FUNCTION_BLOCK FB_Holder
VAR_INPUT
	i_i_HolderPosition:	INT;
	Loaded:BOOL;
	Eingeschraubt	:	BOOL;
	Abgeschraubt: BOOL;
	Nagel: FB_Nagel;
END_VAR

METHOD MoveForward : BOOL
VAR_INPUT

END_VAR
i_i_HolderPosition:=i_i_HolderPosition+1;
END_METHOD

END_FUNCTION_BLOCK

(* stored: Version 1.1.0.1, ProductVersion 3.1.4024.3
   POU FB_Holder: Id {bdc5e698-34c8-4813-aa4a-5c82638240b4}, SpecialFunc None
   Method MoveForward: Id {778157c4-842c-4e24-ba3a-db3c00aa90f1} *)
